INTERFACE ITF_ControlElement_HMI

END_INTERFACE

(* stored: Version 1.1.0.1, ProductVersion 3.1.4024.15
   Itf ITF_ControlElement_HMI: Id {9ab225a5-6d3a-489a-8f21-bf97c3be3e87} *)
